FUNCTION_BLOCK "RateLimiter"
{ S7_Optimized_Access := 'TRUE' }
VERSION : 0.1
   VAR_INPUT
      target : Real;   // AI输出目标值
      maxRateUp : Real := 5.0;   //  最大上升速率（单位/秒）
      maxRateDown : Real := 5.0;   // 最大下降速率（单位/秒），
      cycleTime : Real := 0.01;   // OB1扫描周期（秒），通常 5~15ms
      enable : Bool := TRUE;   // 斜坡使能
      reset : Bool;   // 复位：输出立即跳变到 target
   END_VAR

   VAR_OUTPUT
      output : Real;   // 平滑后的输出值
      isLimited : Bool;   // TRUE = 正在限幅（被斜坡钳制）
   END_VAR

   VAR
      lastOutput : Real;   // 上周期输出值（静态保持）
      initDone : Bool;   // 初始化完成标志
   END_VAR

   VAR_TEMP
      delta : Real;   // 与目标的偏差
      maxStep : Real;   // 本周期允许的最大步长
   END_VAR


BEGIN
	// ===================================================================
	// RateLimiter — 防震荡物理护盾
	// 将高频跳变的目标值平滑为有限速率的变化曲线，保护物理设备
	// ===================================================================

	// --- 首次调用：避免从 0 跳到目标值的阶跃 ---
	IF NOT #initDone THEN
	    #output := #target;
	    #lastOutput := #target;
	    #initDone := TRUE;
	    #isLimited := FALSE;
	    RETURN;
	END_IF;

	// --- 复位模式 ---
	IF #reset THEN
	    #output := #target;
	    #lastOutput := #target;
	    #isLimited := FALSE;
	    RETURN;
	END_IF;

	// --- 正常斜坡控制 ---
	IF #enable AND #cycleTime > 0.0 THEN
	    #delta := #target - #lastOutput;

	    IF #delta > 0.0 THEN
	        // === 上升方向 ===
	        #maxStep := #maxRateUp * #cycleTime;
	        IF #delta > #maxStep THEN
	            #output := #lastOutput + #maxStep;
	            #isLimited := TRUE;
	        ELSE
	            #output := #target;          // 在允许范围内，直接输出
	            #isLimited := FALSE;
	        END_IF;
	    ELSIF #delta < 0.0 THEN
	        // === 下降方向 ===
	        #maxStep := #maxRateDown * #cycleTime;
	        IF - #delta > #maxStep THEN        // 取绝对值比较
	            #output := #lastOutput - #maxStep;
	            #isLimited := TRUE;
	        ELSE
	            #output := #target;
	            #isLimited := FALSE;
	        END_IF;
	    ELSE
	        // delta = 0，目标未变化
	        #output := #target;
	        #isLimited := FALSE;
	    END_IF;
	ELSE
	    // 斜坡禁用或周期无效 — 直通模式
	    #output := #target;
	    #isLimited := FALSE;
	END_IF;

	// --- 保存本周期的输出，供下周期使用 ---
	#lastOutput := #output;
END_FUNCTION_BLOCK

DATA_BLOCK "inst_RL_A"
{ S7_Optimized_Access := 'TRUE' }
VERSION : 0.1
NON_RETAIN
"RateLimiter"

BEGIN

END_DATA_BLOCK

DATA_BLOCK "inst_RL_F"
{ S7_Optimized_Access := 'TRUE' }
VERSION : 0.1
NON_RETAIN
"RateLimiter"

BEGIN

END_DATA_BLOCK

DATA_BLOCK "DB1"
{ DB_Accessible_From_OPC_UA := 'FALSE' ;
 S7_Optimized_Access := 'FALSE' }
VERSION : 0.1
NON_RETAIN
   STRUCT
      // Python/SAC -> PLC. 地址需要和 config/simulation.yaml 保持一致。
      EC_Set_SP : Real;   // DBD0，SAC 输出的目标 EC
      pH_Set_SP : Real;   // DBD4，SAC 输出的目标 pH
      EC_Actual : Real;   // DBD8，Python/传感器反馈的出口 EC
      pH_Actual : Real;   // DBD12，Python/传感器反馈的出口 pH
      SAC_Enable : Bool;   // DBX16.0，远程/SAC 控制使能
      Reserved_17 : Byte;   // DBB17，占位，保证 Remote_Heartbeat 位于 DBW18
      Remote_Heartbeat : Int;
      Remote_Comms_OK : Bool;   // DBX20.0，PLC 判断 Python 通讯是否正常
      Reserved_21 : Byte;   // DBB21，占位，保证 Watchdog_Timer 位于 DBW22
      Watchdog_Timer : Int;
      q_f_cmd : Real;   // DBD24，PLC 输出肥料母液流量 L/min
      q_a_cmd : Real;   // DBD28，PLC 输出酸液流量 L/min
      Valve_F_Actual : Real;   // DBD32，肥液执行量反馈
      Valve_A_Actual : Real;   // DBD36，酸液执行量反馈
      AQ_Valve_F_Raw : Int;
      AQ_Valve_A_Raw : Int;
      System_Alarm_Light : Bool;

      // 以下为 PLC 内部状态，不建议 Python 直接读写。
      Last_Heartbeat : Int;
      Watchdog_Count : Int;
      q_f_raw : Real;
      q_a_raw : Real;
      q_f_limited : Bool;
      q_a_limited : Bool;

      // 兼容旧 A 方案/旧 OB1 网络的变量。放在 Python 固定读写区之后，
      // 不影响 EC_Set_SP、q_f_cmd 等前 45 字节地址。
      Valve_F_Opt_SP : Real;
      Valve_A_Opt_SP : Real;
      Ramp_Target_F : Real;
      Ramp_Target_A : Real;
      Ramp_Step : Real;
      Remote_Comms_Was_OK : Bool;
      Actual_Valve_F : Real;
      Actual_Valve_A : Real;
      tWatchdog {InstructionName := 'TON_TIME'; LibVersion := '1.0'; S7_SetPoint := 'False'} : TON_TIME;
      Growth_Stage : Int;   // 0=INI, 1=DEV, 2=MID, 3=LATE
      Stage_EC_SP : Real;   // 当前生长阶段固定 EC 保护值
      Stage_pH_SP : Real;   // 当前生长阶段固定 pH 保护值
      Active_EC_SP : Real;   // PLC 实际采用的 EC 目标
      Active_pH_SP : Real;   // PLC 实际采用的 pH 目标
      Setpoint_Protection_Active : Bool;   // SAC 目标越界时置 TRUE
      Stage_Auto_SP_Enable : Bool;   // TRUE=PLC 根据 Growth_Stage 自动写 EC_Set_SP/pH_Set_SP

      // PID 在线调参区。Python 粗调或 TIA 监控表可直接写这些值。
      Kp_EC_Set : Real;   // EC 比例增益
      Ki_EC_Set : Real;   // EC 积分增益
      Kd_EC_Set : Real;   // EC 微分增益
      Kp_pH_Set : Real;   // pH 比例增益
      Ki_pH_Set : Real;   // pH 积分增益
      Kd_pH_Set : Real;   // pH 微分增益

      // 多肥液通道在线配置区。Enable 使用 Real(>=0.5 启用)，便于 Snap7 按 DBD 写入。
      N_Enable : Real;      // 氮肥通道启用
      N_Ratio : Real;       // 总肥液 q_f_cmd 分配比例
      N_Target : Real;      // 可选氮目标；无在线 N 传感器时保持 0
      N_Actual : Real;      // 可选氮反馈；无在线 N 传感器时保持 0
      Kp_N_Set : Real;
      Ki_N_Set : Real;
      Kd_N_Set : Real;
      N_Max : Real;
      q_n_cmd : Real;       // 氮肥计量泵输出 L/min
      AQ_Valve_N_Raw : Int;
      N_Reserved : Int;

      P_Enable : Real;      // 磷肥通道启用
      P_Ratio : Real;
      P_Target : Real;
      P_Actual : Real;
      Kp_P_Set : Real;
      Ki_P_Set : Real;
      Kd_P_Set : Real;
      P_Max : Real;
      q_p_cmd : Real;       // 磷肥计量泵输出 L/min
      AQ_Valve_P_Raw : Int;
      P_Reserved : Int;

      K_Enable : Real;      // 钾肥通道启用
      K_Ratio : Real;
      K_Target : Real;
      K_Actual : Real;
      Kp_K_Set : Real;
      Ki_K_Set : Real;
      Kd_K_Set : Real;
      K_Max : Real;
      q_k_cmd : Real;       // 钾肥计量泵输出 L/min
      AQ_Valve_K_Raw : Int;
      K_Reserved : Int;

      // PLC 细调窗口：PID 只允许在前馈流量基础上做有限百分比修正。
      // 推荐范围 0.05~0.15；0.10 表示 EC 肥液输出允许 ±10% 修正。
      EC_Trim_Band : Real;
      pH_Trim_Band : Real;

      // 试验台本地模式区。放在现有 Python 固定地址区之后，避免改变既有 offset。
      Manual_Mode : Bool;       // TRUE=手动调试模式，绕过 EC/pH 自动闭环
      Auto_Mode : Bool;         // TRUE=预留本地自动模式，当前自动仍由 SAC_Enable 驱动
      Emergency_Stop : Bool;    // TRUE=急停，所有执行量立即归零
      Manual_Active : Bool;     // PLC 当前处于手动输出
      Auto_Active : Bool;       // PLC 当前处于自动闭环输出
      Reserved_279 : Byte;      // 占位，使 Manual_q_* 从 DBD280 开始
      Manual_q_f_Set : Real;    // 手动总肥液流量 L/min，限幅 0~10
      Manual_q_a_Set : Real;    // 手动酸液流量 L/min，限幅 0~4
      Manual_q_n_Set : Real;    // 手动氮肥通道 L/min，限幅 0~N_Max
      Manual_q_p_Set : Real;    // 手动磷肥通道 L/min，限幅 0~P_Max
      Manual_q_k_Set : Real;    // 手动钾肥通道 L/min，限幅 0~K_Max

      // LAD 离散联锁与手动输出选择区。从 DBX300/DBD304 继续追加，不改变既有地址。
      Comm_Normal : Bool;              // LAD 判断通信可用：Remote_Comms_OK 且未急停
      Manual_PumpValve_Enable : Bool;  // LAD 手动泵阀使能：Manual_Active 且通信正常
      Reserved_300 : Byte;             // 占位，使手动选择输出从 DBD304 开始
      Reserved_301 : Word;             // 对齐占位
      Manual_q_f_Selected : Real;      // LAD 选择后的手动肥液流量设定
      Manual_q_a_Selected : Real;      // LAD 选择后的手动酸液流量设定
   END_STRUCT;


BEGIN
   EC_Set_SP := 1.5;
   pH_Set_SP := 6.0;
   EC_Actual := 0.0;
   pH_Actual := 7.0;
   SAC_Enable := false;
   Remote_Comms_OK := false;
   q_f_cmd := 0.0;
   q_a_cmd := 0.0;
   Valve_F_Actual := 0.0;
   Valve_A_Actual := 0.0;
   AQ_Valve_F_Raw := 0;
   AQ_Valve_A_Raw := 0;
   System_Alarm_Light := false;
   Valve_F_Opt_SP := 0.0;
   Valve_A_Opt_SP := 0.0;
   Ramp_Target_F := 0.0;
   Ramp_Target_A := 0.0;
   Ramp_Step := 0.0;
   Remote_Comms_Was_OK := false;
   Actual_Valve_F := 0.0;
   Actual_Valve_A := 0.0;
   Growth_Stage := 2;
   Stage_EC_SP := 1.5;
   Stage_pH_SP := 5.9;
   Active_EC_SP := 1.5;
   Active_pH_SP := 5.9;
   Setpoint_Protection_Active := false;
   Stage_Auto_SP_Enable := true;
   Kp_EC_Set := 1.20;
   Ki_EC_Set := 0.0;
   Kd_EC_Set := 0.0;
   Kp_pH_Set := 1.20;
   Ki_pH_Set := 0.01;
   Kd_pH_Set := 0.0;
   N_Enable := 1.0;
   N_Ratio := 0.3333;
   N_Target := 0.0;
   N_Actual := 0.0;
   Kp_N_Set := 0.0;
   Ki_N_Set := 0.0;
   Kd_N_Set := 0.0;
   N_Max := 4.0;
   q_n_cmd := 0.0;
   AQ_Valve_N_Raw := 0;
   N_Reserved := 0;
   P_Enable := 1.0;
   P_Ratio := 0.3333;
   P_Target := 0.0;
   P_Actual := 0.0;
   Kp_P_Set := 0.0;
   Ki_P_Set := 0.0;
   Kd_P_Set := 0.0;
   P_Max := 4.0;
   q_p_cmd := 0.0;
   AQ_Valve_P_Raw := 0;
   P_Reserved := 0;
   K_Enable := 1.0;
   K_Ratio := 0.3334;
   K_Target := 0.0;
   K_Actual := 0.0;
   Kp_K_Set := 0.0;
   Ki_K_Set := 0.0;
   Kd_K_Set := 0.0;
   K_Max := 4.0;
   q_k_cmd := 0.0;
   AQ_Valve_K_Raw := 0;
   K_Reserved := 0;
   EC_Trim_Band := 0.10;
   pH_Trim_Band := 0.08;
   Manual_Mode := false;
   Auto_Mode := true;
   Emergency_Stop := false;
   Manual_Active := false;
   Auto_Active := false;
   Manual_q_f_Set := 0.0;
   Manual_q_a_Set := 0.0;
   Manual_q_n_Set := 0.0;
   Manual_q_p_Set := 0.0;
   Manual_q_k_Set := 0.0;
   Comm_Normal := false;
   Manual_PumpValve_Enable := false;
   Reserved_300 := 0;
   Reserved_301 := 0;
   Manual_q_f_Selected := 0.0;
   Manual_q_a_Selected := 0.0;

END_DATA_BLOCK

FUNCTION_BLOCK "FB_FertigationControl"
{ S7_Optimized_Access := 'TRUE' }
VERSION : 0.1
   VAR_INPUT
      EC_Set_SP : Real;   // 上位机/SAC 目标 EC
      pH_Set_SP : Real;   // 上位机/SAC 目标 pH
      EC_Actual : Real;   // 出口 EC 反馈
      pH_Actual : Real;   // 出口 pH 反馈
      SAC_Enable : Bool;   // 远程控制使能
      Remote_Heartbeat : Int;   // 上位机心跳
      CycleTime : Real := 0.1;   // 调用周期，单位 s
      Kp_EC : Real := 1.20;   // EC PID 比例增益
      Ki_EC : Real := 0.0;   // EC 积分先关闭，避免到目标后继续累积导致过冲
      Kd_EC : Real := 0.0;   // EC PID 微分增益，联调初期先置 0
      Kp_pH : Real := 1.20;   // pH PID 比例增益，pH 偏高时加酸
      Ki_pH : Real := 0.01;   // pH PID 积分增益
      Kd_pH : Real := 0.0;   // pH PID 微分增益，联调初期先置 0
      EC_Filter_Tau : Real := 2.0;   // EC 反馈滤波时间常数，单位 s，越大越稳但响应越慢
      pH_Filter_Tau : Real := 2.0;   // pH 反馈滤波时间常数，单位 s
      EC_Deadband : Real := 0.03;   // EC 小误差死区，避免输出在目标附近来回跳
      pH_Deadband : Real := 0.04;   // pH 小误差死区
      EC_Trim_Band : Real := 0.10;   // PLC 细调窗口，限制 EC PID 在前馈基础上 ±5%~±15%
      pH_Trim_Band : Real := 0.08;   // PLC 细调窗口，限制 pH PID 在前馈基础上 ±5%~±15%
      EC_MaxInputStep : Real := 0.15;   // 每周期允许进入滤波器的最大 EC 跳变
      pH_MaxInputStep : Real := 0.15;   // 每周期允许进入滤波器的最大 pH 跳变
      q_f_min : Real := 0.0;
      q_f_max : Real := 10.0;
      q_a_min : Real := 0.0;
      q_a_max : Real := 4.0;
      N_Enable : Real := 1.0;
      N_Ratio : Real := 0.3333;
      N_Target : Real := 0.0;
      N_Actual : Real := 0.0;
      Kp_N : Real := 0.0;
      Ki_N : Real := 0.0;
      Kd_N : Real := 0.0;
      N_Max : Real := 4.0;
      P_Enable : Real := 1.0;
      P_Ratio : Real := 0.3333;
      P_Target : Real := 0.0;
      P_Actual : Real := 0.0;
      Kp_P : Real := 0.0;
      Ki_P : Real := 0.0;
      Kd_P : Real := 0.0;
      P_Max : Real := 4.0;
      K_Enable : Real := 1.0;
      K_Ratio : Real := 0.3334;
      K_Target : Real := 0.0;
      K_Actual : Real := 0.0;
      Kp_K : Real := 0.0;
      Ki_K : Real := 0.0;
      Kd_K : Real := 0.0;
      K_Max : Real := 4.0;
      Watchdog_Limit : Int := 10000;   // 心跳超限后进入安全输出，需大于两次 Python 写入间隔内的 OB1 扫描次数
      Growth_Stage : Int := 2;   // 0=INI, 1=DEV, 2=MID, 3=LATE
   END_VAR

   VAR_OUTPUT
      Remote_Comms_OK : Bool;
      Watchdog_Timer : Int;
      Stage_EC_SP : Real;
      Stage_pH_SP : Real;
      Active_EC_SP : Real;
      Active_pH_SP : Real;
      Setpoint_Protection_Active : Bool;
      q_f_cmd : Real;
      q_a_cmd : Real;
      Valve_F_Actual : Real;
      Valve_A_Actual : Real;
      AQ_Valve_F_Raw : Int;
      AQ_Valve_A_Raw : Int;
      q_n_cmd : Real;
      q_p_cmd : Real;
      q_k_cmd : Real;
      AQ_Valve_N_Raw : Int;
      AQ_Valve_P_Raw : Int;
      AQ_Valve_K_Raw : Int;
      System_Alarm_Light : Bool;
   END_VAR

   VAR
      Last_Heartbeat : Int;
      Watchdog_Count : Int;
      q_f_raw : Real;
      q_a_raw : Real;
      EC_Integral : Real;
      pH_Integral : Real;
      N_Integral : Real;
      P_Integral : Real;
      K_Integral : Real;
      EC_Error_Last : Real;
      pH_Error_Last : Real;
      N_Error_Last : Real;
      P_Error_Last : Real;
      K_Error_Last : Real;
      Active_EC_SP_Last : Real;
      Active_pH_SP_Last : Real;
      Setpoint_Track_Init : Bool;
      Setpoint_Age_S : Real;
      SAC_Enable_Last : Bool;
      EC_Filtered : Real;
      pH_Filtered : Real;
      Filter_Init : Bool;
      inst_CommsWatchdog : "FB_CommsWatchdog_LAD";
      inst_RL_F : "RateLimiter";
      inst_RL_A : "RateLimiter";
      tWatchdog {InstructionName := 'TON_TIME'; LibVersion := '1.0'; S7_SetPoint := 'False'} : TON_TIME;
   END_VAR

   VAR_TEMP
      EC_Error : Real;
      pH_Error : Real;
      q_f_target : Real;
      q_a_target : Real;
      q_f_feedforward : Real;
      q_f_correction : Real;
      q_a_feedforward : Real;
      q_a_correction : Real;
      Heartbeat_Changed : Bool;
      EC_Derivative : Real;
      pH_Derivative : Real;
      q_f_pid : Real;
      q_a_pid : Real;
      EC_Alpha : Real;
      pH_Alpha : Real;
      EC_InputDelta : Real;
      pH_InputDelta : Real;
      EC_FilterTarget : Real;
      pH_FilterTarget : Real;
      Stage_EC_Min : Real;
      Stage_EC_Max : Real;
      Stage_pH_Min : Real;
      Stage_pH_Max : Real;
      EC_Error_Norm : Real;
      EC_Derivative_Norm : Real;
      pH_Error_Norm : Real;
      pH_Derivative_Norm : Real;
      Kp_EC_Eff : Real;
      Ki_EC_Eff : Real;
      Kd_EC_Eff : Real;
      Kp_pH_Eff : Real;
      Ki_pH_Eff : Real;
      Kd_pH_Eff : Real;
      Setpoint_Changed : Bool;
      q_f_nominal : Real;
      pH_H_Set : Real;
      pH_H_Water : Real;
      pH_H_Acid : Real;
      pH_Denom : Real;
      Feedforward_Only : Bool;
      pH_NearFactor : Real;
      EC_Trim_Band_Safe : Real;
      pH_Trim_Band_Safe : Real;
      q_f_trim_span : Real;
      q_a_trim_span : Real;
      q_f_trim_min : Real;
      q_f_trim_max : Real;
      q_a_trim_min : Real;
      q_a_trim_max : Real;
      N_Error : Real;
      P_Error : Real;
      K_Error : Real;
      N_Derivative : Real;
      P_Derivative : Real;
      K_Derivative : Real;
      q_n_target : Real;
      q_p_target : Real;
      q_k_target : Real;
      q_npk_sum : Real;
      q_npk_scale : Real;
   END_VAR

BEGIN
   // ================================================================
   // B 方案 PLC 执行层
   // Python/SAC 只给 EC_set、pH_set；PLC 根据反馈计算 q_f、q_a。
   // 当前版本为“前馈 + 模糊自适应 PID + 长管道提前停酸/保前馈”。
   // ================================================================

   // --- 心跳监控 ---
   // Python 每次写入都会递增 Remote_Heartbeat；PLC 看到变化则认为通信正常。
   // 这里直接在执行层实现，避免外部 LAD 看门狗未下载或未刷新时锁死输出。
   #Heartbeat_Changed := #Remote_Heartbeat <> #Last_Heartbeat;

   IF #Heartbeat_Changed THEN
      #Last_Heartbeat := #Remote_Heartbeat;
      #Watchdog_Count := 0;
      #Remote_Comms_OK := TRUE;
   ELSE
      IF #Watchdog_Count < #Watchdog_Limit THEN
         #Watchdog_Count := #Watchdog_Count + 1;
      END_IF;
      #Remote_Comms_OK := #Watchdog_Count < #Watchdog_Limit;
   END_IF;

   #Watchdog_Timer := #Watchdog_Count;

   // --- 生长阶段固定目标保护 ---
   // 0=INI 出苗期，1=DEV 营养/形成期，2=MID 膨大期，3=LATE 后期/成熟期。
   IF #Growth_Stage = 0 THEN
      #Stage_EC_SP := 0.8;
      #Stage_pH_SP := 6.2;
      #Stage_EC_Min := 0.7;
      #Stage_EC_Max := 0.9;
      #Stage_pH_Min := 6.1;
      #Stage_pH_Max := 6.3;
   ELSIF #Growth_Stage = 1 THEN
      #Stage_EC_SP := 1.1;
      #Stage_pH_SP := 6.1;
      #Stage_EC_Min := 0.9;
      #Stage_EC_Max := 1.3;
      #Stage_pH_Min := 6.0;
      #Stage_pH_Max := 6.2;
   ELSIF #Growth_Stage = 2 THEN
      #Stage_EC_SP := 1.5;
      #Stage_pH_SP := 5.9;
      #Stage_EC_Min := 1.3;
      #Stage_EC_Max := 1.7;
      #Stage_pH_Min := 5.8;
      #Stage_pH_Max := 6.1;
   ELSE
      #Stage_EC_SP := 1.0;
      #Stage_pH_SP := 6.1;
      #Stage_EC_Min := 0.8;
      #Stage_EC_Max := 1.2;
      #Stage_pH_Min := 6.0;
      #Stage_pH_Max := 6.3;
   END_IF;

   #Active_EC_SP := #EC_Set_SP;
   #Active_pH_SP := #pH_Set_SP;
   #Setpoint_Protection_Active := FALSE;

   IF (#EC_Set_SP < #Stage_EC_Min) OR (#EC_Set_SP > #Stage_EC_Max) THEN
      #Active_EC_SP := #Stage_EC_SP;
      #Setpoint_Protection_Active := TRUE;
   END_IF;

   IF (#pH_Set_SP < #Stage_pH_Min) OR (#pH_Set_SP > #Stage_pH_Max) THEN
      #Active_pH_SP := #Stage_pH_SP;
      #Setpoint_Protection_Active := TRUE;
   END_IF;

   // --- 目标值变化处理 ---
   // 手动或 SAC 改目标时，旧积分和上一误差会把 PID 带偏，导致 EC/pH 大幅摆动。
   // 目标一变化就清掉动态记忆，但保留反馈滤波状态。
   IF NOT #Setpoint_Track_Init THEN
      #Active_EC_SP_Last := #Active_EC_SP;
      #Active_pH_SP_Last := #Active_pH_SP;
      #Setpoint_Track_Init := TRUE;
   END_IF;

   // 只把真正的阶段切换/人工大改目标当作 Setpoint_Changed。
   // 连续小步逼近目标会反复清积分和进入 Feedforward_Only，导致 PID 执行量跳动。
   #Setpoint_Changed := (ABS(#Active_EC_SP - #Active_EC_SP_Last) > 0.05)
      OR (ABS(#Active_pH_SP - #Active_pH_SP_Last) > 0.03);

   IF #SAC_Enable AND NOT #SAC_Enable_Last THEN
      #Setpoint_Changed := TRUE;
   END_IF;

   IF #Setpoint_Changed THEN
      #EC_Integral := 0.0;
      #pH_Integral := 0.0;
      #EC_Error_Last := 0.0;
      #pH_Error_Last := 0.0;
      #Setpoint_Age_S := 0.0;
      #Active_EC_SP_Last := #Active_EC_SP;
      #Active_pH_SP_Last := #Active_pH_SP;
   ELSIF #Heartbeat_Changed THEN
      IF #Setpoint_Age_S < 1200.0 THEN
         #Setpoint_Age_S := #Setpoint_Age_S + 1.0;
      END_IF;
   END_IF;

   // --- 安全状态：未使能或通讯超时，所有执行量归零 ---
   IF (NOT #SAC_Enable) OR (NOT #Remote_Comms_OK) THEN
      #SAC_Enable_Last := FALSE;
      #q_f_raw := 0.0;
      #q_a_raw := 0.0;
      #q_f_cmd := 0.0;
      #q_a_cmd := 0.0;
      #q_n_cmd := 0.0;
      #q_p_cmd := 0.0;
      #q_k_cmd := 0.0;
      #Valve_F_Actual := 0.0;
      #Valve_A_Actual := 0.0;
      #AQ_Valve_F_Raw := 0;
      #AQ_Valve_A_Raw := 0;
      #AQ_Valve_N_Raw := 0;
      #AQ_Valve_P_Raw := 0;
      #AQ_Valve_K_Raw := 0;
      #System_Alarm_Light := NOT #Remote_Comms_OK;
      RETURN;
   END_IF;

   #SAC_Enable_Last := TRUE;

   // --- 反馈滤波 ---
   // Python/传感器写入的 EC_Actual、pH_Actual 可能有瞬时抖动；
   // PID 使用滤波后的值，避免泵阀跟着噪声频繁调整。
   IF NOT #Filter_Init THEN
      #EC_Filtered := #EC_Actual;
      #pH_Filtered := #pH_Actual;
      #Filter_Init := TRUE;
   END_IF;

   IF (#CycleTime > 0.0) AND (#EC_Filter_Tau > 0.0) THEN
      #EC_Alpha := #CycleTime / (#EC_Filter_Tau + #CycleTime);
   ELSE
      #EC_Alpha := 1.0;
   END_IF;

   IF (#CycleTime > 0.0) AND (#pH_Filter_Tau > 0.0) THEN
      #pH_Alpha := #CycleTime / (#pH_Filter_Tau + #CycleTime);
   ELSE
      #pH_Alpha := 1.0;
   END_IF;

   // 基本量程保护 + 输入跳变限制：明显不合理或过快的变化不直接进入滤波器。
   IF (#EC_Actual >= 0.0) AND (#EC_Actual <= 10.0) THEN
      #EC_InputDelta := #EC_Actual - #EC_Filtered;
      IF #EC_InputDelta > #EC_MaxInputStep THEN
         #EC_FilterTarget := #EC_Filtered + #EC_MaxInputStep;
      ELSIF #EC_InputDelta < -#EC_MaxInputStep THEN
         #EC_FilterTarget := #EC_Filtered - #EC_MaxInputStep;
      ELSE
         #EC_FilterTarget := #EC_Actual;
      END_IF;
      #EC_Filtered := #EC_Filtered + #EC_Alpha * (#EC_FilterTarget - #EC_Filtered);
   END_IF;

   IF (#pH_Actual >= 0.0) AND (#pH_Actual <= 14.0) THEN
      #pH_InputDelta := #pH_Actual - #pH_Filtered;
      IF #pH_InputDelta > #pH_MaxInputStep THEN
         #pH_FilterTarget := #pH_Filtered + #pH_MaxInputStep;
      ELSIF #pH_InputDelta < -#pH_MaxInputStep THEN
         #pH_FilterTarget := #pH_Filtered - #pH_MaxInputStep;
      ELSE
         #pH_FilterTarget := #pH_Actual;
      END_IF;
      #pH_Filtered := #pH_Filtered + #pH_Alpha * (#pH_FilterTarget - #pH_Filtered);
   END_IF;

   // --- PID 闭环控制 ---
   // EC 偏低：增加肥料母液流量；EC 偏高：减少肥料母液流量。
   #EC_Error := #Active_EC_SP - #EC_Filtered;

   // pH 偏高：增加酸液流量；pH 偏低：减少酸液流量。
   #pH_Error := #pH_Filtered - #Active_pH_SP;

   IF ABS(#EC_Error) < #EC_Deadband THEN
      #EC_Error := 0.0;
   END_IF;

   IF ABS(#pH_Error) < #pH_Deadband THEN
      #pH_Error := 0.0;
   END_IF;

   IF #CycleTime > 0.0 THEN
      #EC_Integral := #EC_Integral + #EC_Error * #CycleTime;
      #pH_Integral := #pH_Integral + #pH_Error * #CycleTime;

      #EC_Derivative := (#EC_Error - #EC_Error_Last) / #CycleTime;
      #pH_Derivative := (#pH_Error - #pH_Error_Last) / #CycleTime;
   ELSE
      #EC_Derivative := 0.0;
      #pH_Derivative := 0.0;
   END_IF;

   // 积分限幅，防止长时间饱和后积分过大。
   IF #EC_Integral > 5.0 THEN
      #EC_Integral := 5.0;
   ELSIF #EC_Integral < -5.0 THEN
      #EC_Integral := -5.0;
   END_IF;

   IF #pH_Integral > 5.0 THEN
      #pH_Integral := 5.0;
   ELSIF #pH_Integral < -5.0 THEN
      #pH_Integral := -5.0;
   END_IF;

   // --- 模糊自适应 PID 增益 ---
   // 在线写入的 Kp/Ki/Kd 作为基准增益；PLC 根据误差 e 和误差变化率 de
   // 每个扫描周期计算有效增益。误差大时提高 Kp、抑制 Ki，变化快时提高 Kd。
   #EC_Error_Norm := ABS(#EC_Error) / 0.35;
   IF #EC_Error_Norm > 1.0 THEN
      #EC_Error_Norm := 1.0;
   END_IF;

   #EC_Derivative_Norm := ABS(#EC_Derivative) / 0.20;
   IF #EC_Derivative_Norm > 1.0 THEN
      #EC_Derivative_Norm := 1.0;
   END_IF;

   #Kp_EC_Eff := #Kp_EC * (0.75 + 0.55 * #EC_Error_Norm + 0.20 * #EC_Derivative_Norm);
   #Ki_EC_Eff := #Ki_EC * (1.20 - 0.70 * #EC_Error_Norm - 0.30 * #EC_Derivative_Norm);
   #Kd_EC_Eff := #Kd_EC * (0.60 + 0.30 * #EC_Error_Norm + 0.80 * #EC_Derivative_Norm);

   IF #Ki_EC_Eff < 0.0 THEN
      #Ki_EC_Eff := 0.0;
   END_IF;

   #pH_Error_Norm := ABS(#pH_Error) / 0.45;
   IF #pH_Error_Norm > 1.0 THEN
      #pH_Error_Norm := 1.0;
   END_IF;

   #pH_Derivative_Norm := ABS(#pH_Derivative) / 0.20;
   IF #pH_Derivative_Norm > 1.0 THEN
      #pH_Derivative_Norm := 1.0;
   END_IF;

   #Kp_pH_Eff := #Kp_pH * (0.75 + 0.55 * #pH_Error_Norm + 0.20 * #pH_Derivative_Norm);
   #Ki_pH_Eff := #Ki_pH * (1.20 - 0.70 * #pH_Error_Norm - 0.30 * #pH_Derivative_Norm);
   #Kd_pH_Eff := #Kd_pH * (0.60 + 0.30 * #pH_Error_Norm + 0.80 * #pH_Derivative_Norm);

   IF #Ki_pH_Eff < 0.0 THEN
      #Ki_pH_Eff := 0.0;
   END_IF;

   // 真实管道存在约 8 min 纯滞后。目标刚改变时，反馈仍是旧目标；
   // 此时若让 PID 强修正，会把正确前馈推偏。先用前馈等待管道响应。
   #Feedforward_Only := #Setpoint_Age_S < 60.0;

   // pH 前馈按混合模型连续计算，避免目标 pH 改变时分档前馈偏差过大。
   IF (#Active_EC_SP > 0.0) AND (#Active_EC_SP < 34.0) THEN
      #q_f_nominal := (#Active_EC_SP * 136.0) / (35.0 - #Active_EC_SP);
   ELSE
      #q_f_nominal := 0.0;
   END_IF;

   #pH_H_Set := EXP(-#Active_pH_SP * LN(10.0));
   #pH_H_Water := 6.30957E-8;   // 10^-7.2
   #pH_H_Acid := 1.25893E-4;    // 10^-3.9
   #pH_Denom := #pH_H_Acid - #pH_H_Set;

   IF #pH_Denom > 1.0E-9 THEN
      #q_a_feedforward := (#pH_H_Set * (136.0 + #q_f_nominal) - 136.0 * #pH_H_Water) / #pH_Denom;
   ELSE
      #q_a_feedforward := 0.0;
   END_IF;

   IF #q_a_feedforward < 0.0 THEN
      #q_a_feedforward := 0.0;
   ELSIF #q_a_feedforward > #q_a_max THEN
      #q_a_feedforward := #q_a_max;
   END_IF;

   // EC 平衡前馈 + 模糊 PID 修正：
   // 当前数字孪生清水流量 q_w=136 L/min，肥料母液 EC=35 dS/m。
   // 酸液会稀释 EC，因此 EC 前馈按 q_w + q_a_feedforward 计算。
   IF (#Active_EC_SP > 0.0) AND (#Active_EC_SP < 34.0) THEN
      #q_f_feedforward := (#Active_EC_SP * (136.0 + #q_a_feedforward)) / (35.0 - #Active_EC_SP);
   ELSE
      #q_f_feedforward := 0.0;
   END_IF;

   IF #Feedforward_Only THEN
      #q_f_correction := 0.0;
   ELSIF #EC_Error > 0.03 THEN
      #q_f_correction := #Kp_EC_Eff * #EC_Error + #Ki_EC_Eff * #EC_Integral + #Kd_EC_Eff * #EC_Derivative;
   ELSIF #EC_Error < -0.08 THEN
      #q_f_correction := 3.50 * #EC_Error;
   ELSIF #EC_Error < -0.03 THEN
      #q_f_correction := 2.00 * #EC_Error;
   ELSE
      #q_f_correction := 0.0;
   END_IF;

   #EC_Trim_Band_Safe := #EC_Trim_Band;
   IF #EC_Trim_Band_Safe < 0.05 THEN
      #EC_Trim_Band_Safe := 0.05;
   ELSIF #EC_Trim_Band_Safe > 0.15 THEN
      #EC_Trim_Band_Safe := 0.15;
   END_IF;

   #q_f_trim_span := #q_f_feedforward * #EC_Trim_Band_Safe;
   IF #q_f_correction > #q_f_trim_span THEN
      #q_f_correction := #q_f_trim_span;
   ELSIF #q_f_correction < -#q_f_trim_span THEN
      #q_f_correction := -#q_f_trim_span;
   END_IF;
   #q_f_trim_min := #q_f_feedforward - #q_f_trim_span;
   #q_f_trim_max := #q_f_feedforward + #q_f_trim_span;

   #q_f_pid := #q_f_feedforward + #q_f_correction;

   IF #Feedforward_Only THEN
      #q_a_correction := 0.0;
   ELSIF #pH_Error > 0.45 THEN
      #q_a_correction := #q_a_max;
   ELSIF #pH_Error > 0.25 THEN
      #q_a_correction := 3.20 * #pH_Error + 0.85;
   ELSIF #pH_Error > 0.0 THEN
      #q_a_correction := #Kp_pH_Eff * #pH_Error + #Ki_pH_Eff * #pH_Integral + #Kd_pH_Eff * #pH_Derivative;
   ELSIF #pH_Error < -0.10 THEN
      #q_a_correction := 2.50 * #pH_Error;
   ELSE
      #q_a_correction := 0.0;
   END_IF;

   #pH_Trim_Band_Safe := #pH_Trim_Band;
   IF #pH_Trim_Band_Safe < 0.05 THEN
      #pH_Trim_Band_Safe := 0.05;
   ELSIF #pH_Trim_Band_Safe > 0.15 THEN
      #pH_Trim_Band_Safe := 0.15;
   END_IF;

   #q_a_trim_span := #q_a_feedforward * #pH_Trim_Band_Safe;
   IF #q_a_correction > #q_a_trim_span THEN
      #q_a_correction := #q_a_trim_span;
   ELSIF #q_a_correction < -#q_a_trim_span THEN
      #q_a_correction := -#q_a_trim_span;
   END_IF;
   #q_a_trim_min := #q_a_feedforward - #q_a_trim_span;
   #q_a_trim_max := #q_a_feedforward + #q_a_trim_span;

   #q_a_pid := #q_a_feedforward + #q_a_correction;

   #q_f_target := #q_f_pid;
   #q_a_target := #q_a_pid;

   #EC_Error_Last := #EC_Error;
   #pH_Error_Last := #pH_Error;

   // --- EC 超调保护：明显高于目标时必须停肥 ---
   // 目标附近优先保持前馈维持量；但 EC 已经高出较多时继续给前馈会越调越高。
   IF (NOT #Feedforward_Only) AND (#EC_Filtered > (#Active_EC_SP + 0.12)) THEN
      #q_f_target := 0.0;
      #EC_Integral := 0.0;
   ELSIF (NOT #Feedforward_Only) AND (#EC_Filtered > (#Active_EC_SP + 0.06)) THEN
      #q_f_target := 0.0;
      #EC_Integral := 0.0;
   ELSIF (NOT #Feedforward_Only) AND (#EC_Filtered >= (#Active_EC_SP - 0.01)) THEN
      #q_f_target := #q_f_feedforward;
      #EC_Integral := 0.0;
   END_IF;

   // pH 的执行方向相反：加酸会降低 pH。
   // pH 已经低于目标时必须停酸；目标附近才允许维持前馈，避免继续下探。
   IF (NOT #Feedforward_Only) AND (#pH_Filtered <= (#Active_pH_SP - 0.08)) THEN
      #q_a_target := 0.0;
      #pH_Integral := 0.0;
   ELSIF (NOT #Feedforward_Only) AND (#pH_Filtered <= (#Active_pH_SP - 0.04)) THEN
      #pH_NearFactor := (#pH_Filtered - (#Active_pH_SP - 0.08)) / 0.04;
      IF #pH_NearFactor < 0.0 THEN
         #pH_NearFactor := 0.0;
      ELSIF #pH_NearFactor > 1.0 THEN
         #pH_NearFactor := 1.0;
      END_IF;
      #q_a_target := #q_a_feedforward * #pH_NearFactor;
      #pH_Integral := 0.0;
   ELSIF (NOT #Feedforward_Only) AND (#pH_Filtered <= (#Active_pH_SP + 0.08)) THEN
      #q_a_target := #q_a_feedforward;
      #pH_Integral := 0.0;
   END_IF;

   // 最终保险：上限锁在前馈窗口内，下限允许到 0，用于超调后的停肥/停酸。
   IF #q_f_target > #q_f_trim_max THEN
      #q_f_target := #q_f_trim_max;
   END_IF;

   IF #q_a_target > #q_a_trim_max THEN
      #q_a_target := #q_a_trim_max;
   END_IF;

   // --- 物理限幅 ---
   IF #q_f_target < #q_f_min THEN
      #q_f_target := #q_f_min;
   ELSIF #q_f_target > #q_f_max THEN
      #q_f_target := #q_f_max;
   END_IF;

   IF #q_a_target < #q_a_min THEN
      #q_a_target := #q_a_min;
   ELSIF #q_a_target > #q_a_max THEN
      #q_a_target := #q_a_max;
   END_IF;

   // --- 斜坡限速，保护泵阀 ---
   #inst_RL_F(
      target := #q_f_target,
      maxRateUp := 1.5,
      maxRateDown := 2.0,
      cycleTime := #CycleTime,
      enable := TRUE,
      reset := FALSE
   );

   #inst_RL_A(
      target := #q_a_target,
      maxRateUp := 0.40,
      maxRateDown := 0.45,
      cycleTime := #CycleTime,
      enable := TRUE,
      reset := FALSE
   );

   #q_f_cmd := #inst_RL_F.output;
   #q_a_cmd := #inst_RL_A.output;
   #q_f_raw := #q_f_cmd;
   #q_a_raw := #q_a_cmd;

   // --- 多肥液通道分配 ---
   // q_f_cmd 保留为“总肥液需求”，N/P/K 三路按 Ratio 分配。
   // 若后续接入在线 N/P/K 传感器，可通过 Target/Actual + PID 对单通道微调。
   IF #CycleTime > 0.0 THEN
      #N_Error := #N_Target - #N_Actual;
      #P_Error := #P_Target - #P_Actual;
      #K_Error := #K_Target - #K_Actual;
      #N_Integral := #N_Integral + #N_Error * #CycleTime;
      #P_Integral := #P_Integral + #P_Error * #CycleTime;
      #K_Integral := #K_Integral + #K_Error * #CycleTime;
      #N_Derivative := (#N_Error - #N_Error_Last) / #CycleTime;
      #P_Derivative := (#P_Error - #P_Error_Last) / #CycleTime;
      #K_Derivative := (#K_Error - #K_Error_Last) / #CycleTime;
   ELSE
      #N_Error := 0.0;
      #P_Error := 0.0;
      #K_Error := 0.0;
      #N_Derivative := 0.0;
      #P_Derivative := 0.0;
      #K_Derivative := 0.0;
   END_IF;

   IF #N_Integral > 5.0 THEN
      #N_Integral := 5.0;
   ELSIF #N_Integral < -5.0 THEN
      #N_Integral := -5.0;
   END_IF;
   IF #P_Integral > 5.0 THEN
      #P_Integral := 5.0;
   ELSIF #P_Integral < -5.0 THEN
      #P_Integral := -5.0;
   END_IF;
   IF #K_Integral > 5.0 THEN
      #K_Integral := 5.0;
   ELSIF #K_Integral < -5.0 THEN
      #K_Integral := -5.0;
   END_IF;

   IF #N_Enable >= 0.5 THEN
      #q_n_target := #q_f_cmd * #N_Ratio + #Kp_N * #N_Error + #Ki_N * #N_Integral + #Kd_N * #N_Derivative;
   ELSE
      #q_n_target := 0.0;
      #N_Integral := 0.0;
   END_IF;

   IF #P_Enable >= 0.5 THEN
      #q_p_target := #q_f_cmd * #P_Ratio + #Kp_P * #P_Error + #Ki_P * #P_Integral + #Kd_P * #P_Derivative;
   ELSE
      #q_p_target := 0.0;
      #P_Integral := 0.0;
   END_IF;

   IF #K_Enable >= 0.5 THEN
      #q_k_target := #q_f_cmd * #K_Ratio + #Kp_K * #K_Error + #Ki_K * #K_Integral + #Kd_K * #K_Derivative;
   ELSE
      #q_k_target := 0.0;
      #K_Integral := 0.0;
   END_IF;

   IF #q_n_target < 0.0 THEN
      #q_n_target := 0.0;
   ELSIF #q_n_target > #N_Max THEN
      #q_n_target := #N_Max;
   END_IF;
   IF #q_p_target < 0.0 THEN
      #q_p_target := 0.0;
   ELSIF #q_p_target > #P_Max THEN
      #q_p_target := #P_Max;
   END_IF;
   IF #q_k_target < 0.0 THEN
      #q_k_target := 0.0;
   ELSIF #q_k_target > #K_Max THEN
      #q_k_target := #K_Max;
   END_IF;

   #q_npk_sum := #q_n_target + #q_p_target + #q_k_target;
   IF (#q_npk_sum > #q_f_cmd) AND (#q_npk_sum > 0.0) THEN
      #q_npk_scale := #q_f_cmd / #q_npk_sum;
      #q_n_target := #q_n_target * #q_npk_scale;
      #q_p_target := #q_p_target * #q_npk_scale;
      #q_k_target := #q_k_target * #q_npk_scale;
   END_IF;

   #q_n_cmd := #q_n_target;
   #q_p_cmd := #q_p_target;
   #q_k_cmd := #q_k_target;
   #N_Error_Last := #N_Error;
   #P_Error_Last := #P_Error;
   #K_Error_Last := #K_Error;

   #Valve_F_Actual := #q_f_cmd;
   #Valve_A_Actual := #q_a_cmd;

   // --- 0~27648 模拟量换算 ---
   #AQ_Valve_F_Raw := REAL_TO_INT(#q_f_cmd / #q_f_max * 27648.0);
   #AQ_Valve_A_Raw := REAL_TO_INT(#q_a_cmd / #q_a_max * 27648.0);
   IF #N_Max > 0.0 THEN
      #AQ_Valve_N_Raw := REAL_TO_INT(#q_n_cmd / #N_Max * 27648.0);
   ELSE
      #AQ_Valve_N_Raw := 0;
   END_IF;
   IF #P_Max > 0.0 THEN
      #AQ_Valve_P_Raw := REAL_TO_INT(#q_p_cmd / #P_Max * 27648.0);
   ELSE
      #AQ_Valve_P_Raw := 0;
   END_IF;
   IF #K_Max > 0.0 THEN
      #AQ_Valve_K_Raw := REAL_TO_INT(#q_k_cmd / #K_Max * 27648.0);
   ELSE
      #AQ_Valve_K_Raw := 0;
   END_IF;

   #System_Alarm_Light := FALSE;
END_FUNCTION_BLOCK

DATA_BLOCK "inst_FertigationControl"
{ S7_Optimized_Access := 'TRUE' }
VERSION : 0.1
NON_RETAIN
"FB_FertigationControl"

BEGIN

END_DATA_BLOCK

FUNCTION "FC_CallFertigationControl" : Void
{ S7_Optimized_Access := 'TRUE' }
VERSION : 0.1
   VAR_TEMP
      Manual_q_f_target : Real;
      Manual_q_a_target : Real;
      Manual_q_n_target : Real;
      Manual_q_p_target : Real;
      Manual_q_k_target : Real;
   END_VAR

BEGIN
   // 在 OB1 中调用本 FC，即可完成：
   // DB1 输入区 -> FB_FertigationControl -> DB1 输出区。
   // 优先级：急停 > 手动模式 > 自动闭环。
   // 开关量模式联锁、报警灯和 q_f/q_a 手动选择由 LAD 块完成。
   // 连续量限幅、斜坡、模拟量换算和自动控制算法保留在 SCL。

   "FC_ModeInterlock_LAD"();

   IF "DB1".Emergency_Stop THEN
      "DB1".q_f_cmd := 0.0;
      "DB1".q_a_cmd := 0.0;
      "DB1".q_n_cmd := 0.0;
      "DB1".q_p_cmd := 0.0;
      "DB1".q_k_cmd := 0.0;
      "DB1".Valve_F_Actual := 0.0;
      "DB1".Valve_A_Actual := 0.0;
      "DB1".AQ_Valve_F_Raw := 0;
      "DB1".AQ_Valve_A_Raw := 0;
      "DB1".AQ_Valve_N_Raw := 0;
      "DB1".AQ_Valve_P_Raw := 0;
      "DB1".AQ_Valve_K_Raw := 0;
      "DB1".Actual_Valve_F := 0.0;
      "DB1".Actual_Valve_A := 0.0;
      "DB1".Valve_F_Opt_SP := 0.0;
      "DB1".Valve_A_Opt_SP := 0.0;
      "DB1".Ramp_Target_F := 0.0;
      "DB1".Ramp_Target_A := 0.0;
      RETURN;
   END_IF;

   IF "DB1".Manual_PumpValve_Enable THEN
      #Manual_q_f_target := "DB1".Manual_q_f_Selected;
      IF #Manual_q_f_target < 0.0 THEN
         #Manual_q_f_target := 0.0;
      ELSIF #Manual_q_f_target > 10.0 THEN
         #Manual_q_f_target := 10.0;
      END_IF;

      #Manual_q_a_target := "DB1".Manual_q_a_Selected;
      IF #Manual_q_a_target < 0.0 THEN
         #Manual_q_a_target := 0.0;
      ELSIF #Manual_q_a_target > 4.0 THEN
         #Manual_q_a_target := 4.0;
      END_IF;

      #Manual_q_n_target := "DB1".Manual_q_n_Set;
      IF #Manual_q_n_target < 0.0 THEN
         #Manual_q_n_target := 0.0;
      ELSIF #Manual_q_n_target > "DB1".N_Max THEN
         #Manual_q_n_target := "DB1".N_Max;
      END_IF;

      #Manual_q_p_target := "DB1".Manual_q_p_Set;
      IF #Manual_q_p_target < 0.0 THEN
         #Manual_q_p_target := 0.0;
      ELSIF #Manual_q_p_target > "DB1".P_Max THEN
         #Manual_q_p_target := "DB1".P_Max;
      END_IF;

      #Manual_q_k_target := "DB1".Manual_q_k_Set;
      IF #Manual_q_k_target < 0.0 THEN
         #Manual_q_k_target := 0.0;
      ELSIF #Manual_q_k_target > "DB1".K_Max THEN
         #Manual_q_k_target := "DB1".K_Max;
      END_IF;

      "inst_RL_F"(
         target := #Manual_q_f_target,
         maxRateUp := 1.5,
         maxRateDown := 2.0,
         cycleTime := 0.1,
         enable := TRUE,
         reset := FALSE,
         output => "DB1".q_f_cmd,
         isLimited => "DB1".q_f_limited
      );

      "inst_RL_A"(
         target := #Manual_q_a_target,
         maxRateUp := 0.40,
         maxRateDown := 0.45,
         cycleTime := 0.1,
         enable := TRUE,
         reset := FALSE,
         output => "DB1".q_a_cmd,
         isLimited => "DB1".q_a_limited
      );

      "DB1".q_n_cmd := #Manual_q_n_target;
      "DB1".q_p_cmd := #Manual_q_p_target;
      "DB1".q_k_cmd := #Manual_q_k_target;
      "DB1".q_f_raw := "DB1".q_f_cmd;
      "DB1".q_a_raw := "DB1".q_a_cmd;
      "DB1".Valve_F_Actual := "DB1".q_f_cmd;
      "DB1".Valve_A_Actual := "DB1".q_a_cmd;
      "DB1".AQ_Valve_F_Raw := REAL_TO_INT("DB1".q_f_cmd / 10.0 * 27648.0);
      "DB1".AQ_Valve_A_Raw := REAL_TO_INT("DB1".q_a_cmd / 4.0 * 27648.0);
      IF "DB1".N_Max > 0.0 THEN
         "DB1".AQ_Valve_N_Raw := REAL_TO_INT("DB1".q_n_cmd / "DB1".N_Max * 27648.0);
      ELSE
         "DB1".AQ_Valve_N_Raw := 0;
      END_IF;
      IF "DB1".P_Max > 0.0 THEN
         "DB1".AQ_Valve_P_Raw := REAL_TO_INT("DB1".q_p_cmd / "DB1".P_Max * 27648.0);
      ELSE
         "DB1".AQ_Valve_P_Raw := 0;
      END_IF;
      IF "DB1".K_Max > 0.0 THEN
         "DB1".AQ_Valve_K_Raw := REAL_TO_INT("DB1".q_k_cmd / "DB1".K_Max * 27648.0);
      ELSE
         "DB1".AQ_Valve_K_Raw := 0;
      END_IF;
      "DB1".Actual_Valve_F := "DB1".Valve_F_Actual;
      "DB1".Actual_Valve_A := "DB1".Valve_A_Actual;
      "DB1".Valve_F_Opt_SP := "DB1".q_f_cmd;
      "DB1".Valve_A_Opt_SP := "DB1".q_a_cmd;
      "DB1".Ramp_Target_F := "DB1".q_f_cmd;
      "DB1".Ramp_Target_A := "DB1".q_a_cmd;
      RETURN;
   END_IF;

   IF NOT "DB1".Auto_Active THEN
      "DB1".q_f_cmd := 0.0;
      "DB1".q_a_cmd := 0.0;
      "DB1".q_n_cmd := 0.0;
      "DB1".q_p_cmd := 0.0;
      "DB1".q_k_cmd := 0.0;
      "DB1".Valve_F_Actual := 0.0;
      "DB1".Valve_A_Actual := 0.0;
      "DB1".AQ_Valve_F_Raw := 0;
      "DB1".AQ_Valve_A_Raw := 0;
      "DB1".AQ_Valve_N_Raw := 0;
      "DB1".AQ_Valve_P_Raw := 0;
      "DB1".AQ_Valve_K_Raw := 0;
      "DB1".Actual_Valve_F := 0.0;
      "DB1".Actual_Valve_A := 0.0;
      "DB1".Valve_F_Opt_SP := 0.0;
      "DB1".Valve_A_Opt_SP := 0.0;
      "DB1".Ramp_Target_F := 0.0;
      "DB1".Ramp_Target_A := 0.0;
      RETURN;
   END_IF;

   IF "DB1".Stage_Auto_SP_Enable AND NOT "DB1".SAC_Enable THEN
      IF "DB1".Growth_Stage = 0 THEN
         "DB1".EC_Set_SP := 0.8;
         "DB1".pH_Set_SP := 6.2;
      ELSIF "DB1".Growth_Stage = 1 THEN
         "DB1".EC_Set_SP := 1.1;
         "DB1".pH_Set_SP := 6.1;
      ELSIF "DB1".Growth_Stage = 2 THEN
         "DB1".EC_Set_SP := 1.5;
         "DB1".pH_Set_SP := 5.9;
      ELSE
         "DB1".EC_Set_SP := 1.0;
         "DB1".pH_Set_SP := 6.1;
      END_IF;
   END_IF;

   "inst_FertigationControl"(
      EC_Set_SP := "DB1".EC_Set_SP,
      pH_Set_SP := "DB1".pH_Set_SP,
      EC_Actual := "DB1".EC_Actual,
      pH_Actual := "DB1".pH_Actual,
      SAC_Enable := "DB1".SAC_Enable,
      Remote_Heartbeat := "DB1".Remote_Heartbeat,
      CycleTime := 0.1,
      Kp_EC := "DB1".Kp_EC_Set,
      Ki_EC := "DB1".Ki_EC_Set,
      Kd_EC := "DB1".Kd_EC_Set,
      Kp_pH := "DB1".Kp_pH_Set,
      Ki_pH := "DB1".Ki_pH_Set,
      Kd_pH := "DB1".Kd_pH_Set,
      EC_Filter_Tau := 2.0,
      pH_Filter_Tau := 4.0,
      EC_Deadband := 0.03,
      pH_Deadband := 0.06,
      EC_Trim_Band := "DB1".EC_Trim_Band,
      pH_Trim_Band := "DB1".pH_Trim_Band,
      EC_MaxInputStep := 0.15,
      pH_MaxInputStep := 0.10,
      q_f_min := 0.0,
      q_f_max := 10.0,
      q_a_min := 0.0,
      q_a_max := 4.0,
      N_Enable := "DB1".N_Enable,
      N_Ratio := "DB1".N_Ratio,
      N_Target := "DB1".N_Target,
      N_Actual := "DB1".N_Actual,
      Kp_N := "DB1".Kp_N_Set,
      Ki_N := "DB1".Ki_N_Set,
      Kd_N := "DB1".Kd_N_Set,
      N_Max := "DB1".N_Max,
      P_Enable := "DB1".P_Enable,
      P_Ratio := "DB1".P_Ratio,
      P_Target := "DB1".P_Target,
      P_Actual := "DB1".P_Actual,
      Kp_P := "DB1".Kp_P_Set,
      Ki_P := "DB1".Ki_P_Set,
      Kd_P := "DB1".Kd_P_Set,
      P_Max := "DB1".P_Max,
      K_Enable := "DB1".K_Enable,
      K_Ratio := "DB1".K_Ratio,
      K_Target := "DB1".K_Target,
      K_Actual := "DB1".K_Actual,
      Kp_K := "DB1".Kp_K_Set,
      Ki_K := "DB1".Ki_K_Set,
      Kd_K := "DB1".Kd_K_Set,
      K_Max := "DB1".K_Max,
      Watchdog_Limit := 10000,
      Growth_Stage := "DB1".Growth_Stage,
      Remote_Comms_OK => "DB1".Remote_Comms_OK,
      Watchdog_Timer => "DB1".Watchdog_Timer,
      Stage_EC_SP => "DB1".Stage_EC_SP,
      Stage_pH_SP => "DB1".Stage_pH_SP,
      Active_EC_SP => "DB1".Active_EC_SP,
      Active_pH_SP => "DB1".Active_pH_SP,
      Setpoint_Protection_Active => "DB1".Setpoint_Protection_Active,
      q_f_cmd => "DB1".q_f_cmd,
      q_a_cmd => "DB1".q_a_cmd,
      Valve_F_Actual => "DB1".Valve_F_Actual,
      Valve_A_Actual => "DB1".Valve_A_Actual,
      AQ_Valve_F_Raw => "DB1".AQ_Valve_F_Raw,
      AQ_Valve_A_Raw => "DB1".AQ_Valve_A_Raw,
      q_n_cmd => "DB1".q_n_cmd,
      q_p_cmd => "DB1".q_p_cmd,
      q_k_cmd => "DB1".q_k_cmd,
      AQ_Valve_N_Raw => "DB1".AQ_Valve_N_Raw,
      AQ_Valve_P_Raw => "DB1".AQ_Valve_P_Raw,
      AQ_Valve_K_Raw => "DB1".AQ_Valve_K_Raw
   );

   // 同步部分内部状态到 DB1，方便在线监控。
   "DB1".Last_Heartbeat := "inst_FertigationControl".Last_Heartbeat;
   "DB1".Watchdog_Count := "inst_FertigationControl".Watchdog_Count;
   "DB1".q_f_raw := "inst_FertigationControl".q_f_raw;
   "DB1".q_a_raw := "inst_FertigationControl".q_a_raw;

   // 兼容旧变量名，若旧监控画面或旧网络还在看 Actual_Valve_F/A，
   // 这里同步为当前 B 方案执行层输出。
   "DB1".Actual_Valve_F := "DB1".Valve_F_Actual;
   "DB1".Actual_Valve_A := "DB1".Valve_A_Actual;
   "DB1".Valve_F_Opt_SP := "DB1".q_f_cmd;
   "DB1".Valve_A_Opt_SP := "DB1".q_a_cmd;
   "DB1".Ramp_Target_F := "DB1".q_f_cmd;
   "DB1".Ramp_Target_A := "DB1".q_a_cmd;
   "DB1".Remote_Comms_Was_OK := "DB1".Remote_Comms_OK;
END_FUNCTION

